(* Logix 5000 project; controller Ceca_1650T_Press 5069-L306ERM rev 32.11; software revision 32.02; part 2 of 3 *)
(* tags used below, declared in another part *)
   STATUS_MESSAGE : STRING;
   AUTO_CYCLE_ENABLED : BOOL;   // M0014 HMI SELECTION
   AUTO_LOWER_LIMIT : BOOL;   // ENCODER SIGNAL B0155
   AUTO_ONE_CYCLE_ENABLED : BOOL;   // M0013 HMI SELECTION
   AUTO_RESET_ALLOWED : BOOL;   // M003E
   AUTO_UPPER_LIMIT : BOOL;   // ENCODER SIGNAL B0151
   BLANKING_OFF_SIGNAL : TIMER;   // T0018
   BLANKING_PS_ENABLED : BOOL;   // M0018
   BOLSTER_CLAMP_ON : BOOL;   // M0006
   BOLSTER_IN_LIMIT : BOOL;   // B000E
   BOLSTER_TOUCH_LIMIT_1 : BOOL;   // B0014
   BOLSTER_TOUCH_LIMIT_2 : BOOL;   // B0015
   BOTH_DIE_CUSHIONS_DOWN : BOOL;   // M0036
   CANCEL_CYLINDER_LOWER_LIMIT : BOOL;   // B000A
   DEBOUNCE_TIMER_LOCKING_OFF : TIMER;   // T0005
   DEBOUNCE_TIMER_LOCKING_OFF_COMPLETE : TIMER;   // T0006
   DECOMPRESSION : BOOL;   // M006D
   DIE_CUSHION_2_PAD_SELECT_RL : BOOL;   // M001D
   DIE_CUSHION_PB_OFF_STATE : BOOL;   // M003F
   DIE_DRAWRIC_CYLINDER_UPPER_PS : BOOL;   // B0018
   DIE_DRAWRIC_DECOMPRESSION_VALVE : BOOL;   // B0056
   DIE_DRAWRIC_DOWN : BOOL;   // M004F
   DIE_DRAWRIC_ON_SELECT : BOOL;   // B0145 HMI BUTTON
   DIE_DRAWRIC_POWER_ASSIST_VALVE : BOOL;   // B0057
   DIE_DRAWRIC_UP : BOOL;   // M004E
   DIE_DRAWRIC_UP_1 : BOOL;   // M007E
   DIE_DRAWRIC_UP_COMPLETE : BOOL;   // M007F
   DIE_DRAWRIC_UP_MEM : TIMER;   // T0019
   DRAW_BLANKING_NOT_SELECT : BOOL;   // M0017
   DRAW_UP_ASSIST : BOOL;   // M007C
   DRAW_UP_ASSIST_COMPLETE : BOOL;   // M007D
   DRAWING_LS_ENABLED : BOOL;   // M0016
   ENABLE_1000T : BOOL;   // HMI BUTTON/RECIPE
   ENABLE_1500T : BOOL;   // HMI BUTTON/RECIPE
   ENABLE_500T : BOOL;   // HMI BUTTON/RECIPE
   FILTER_CHOKER : BOOL;   // B001A
   FILTER_CLOGGED_DELAY : TIMER;   // T0003
   FILTER_CLOGGED_FAULT : BOOL;   // M0023
   FRONT_SHUTTER_SAFETY : BOOL;   // M002A
   INCH_ENABLED : BOOL;   // M0012 HMI SELECTION
   INCHING_SELECTED : BOOL;   // HMI BUTTON/SELECTION B0100
   LOCKING_OFF : BOOL;   // M0004
   LOCKING_OFF_ASSIST : BOOL;   // M0032
   LOCKING_OFF_COMPLETE : BOOL;   // M0033
   LOCKING_OFF_LIMIT : BOOL;   // B0007
   LOCKING_OFF_MEMORY : BOOL;   // M0031
   LOCKING_OFF_VALVE : BOOL;   // B0058
   LOCKING_ON : BOOL;   // M0005
   LOCKING_ON_LIMIT : BOOL;   // B0008
   LUBE_LEVEL_DELAY : TIMER;   // T0002
   LUBE_LEVEL_FAULT : BOOL;   // M0022
   LUBRICATION_FAULT : BOOL;   // M0020
   LUBRICATION_OIL_LEVEL_DETECT : BOOL;   // B001F
   LUBRICATION_PRESSURE_DETECT : BOOL;   // B0017
   M_PRESS_DOWN : BOOL;   // M006A
   M_PRESS_DOWN_COMPLETE : BOOL;   // M006C
   M_PRESS_DOWN_COMPLETE_TIMER : TIMER;   // T0012
   M_PRESS_UP : BOOL;   // M006E
   M_PRESS_UP_COMPLETE : BOOL;   // M006F
   MAIN_DOWN_VALVE : BOOL;   // B0041
   MAIN_DOWN_VALVE_1000_TON : BOOL;   // B0043
   MAIN_DOWN_VALVE_500_TON : BOOL;   // B0042
   MAIN_LOWER_ASSIST_LIMIT : BOOL;   // B0026
   MAIN_LOWER_LIMIT : BOOL;   // B0002
   MAIN_NO_LOAD_VALVE : BOOL;   // B0046
   MAIN_POWER_HOLDING_VALVE : BOOL;   // B0045
   MAIN_PRESS_CONDITION_DOWN : BOOL;   // M0039
   MAIN_PRESS_CONDITION_UP : BOOL;   // M0038
   MAIN_PRESS_DOWN : BOOL;   // M0045
   MAIN_PRESS_DOWN_ASSIST : BOOL;   // M0044
   MAIN_PRESS_NO_PRESSURE_DOWN : BOOL;   // M0047
   MAIN_PRESS_PRESSURE_DETECT : BOOL;   // B0016
   MAIN_PRESS_SLOW_DOWN : BOOL;   // M0046
   MAIN_PRESS_SLOW_DOWN_SIGNAL : BOOL;   // M0030
   MAIN_PRESS_SLOW_UP : BOOL;   // M0042
   MAIN_PRESS_UP : BOOL;   // M0041
   MAIN_PRESS_UP_ASSIST : BOOL;   // M0040
   MAIN_SLOW_DOWN_VALVE : BOOL;   // B0044
   MAIN_UP_VALVE : BOOL;   // B0040
   MAIN_UPPER_LIMIT : BOOL;   // B0000
   MOVEMENT_CONFIRMED : BOOL;   // M0064 M0065 M0066
   NO_PRESSUE_DOWN_PB : BOOL;   // B010D HMI BUTTON
   OIL_TEMP_TOO_HIGH : BOOL;   // B0143
   OIL_TEMPERATURE_FAULT : BOOL;   // M0025
   OIL_WORKING_LEVEL_FAULT : BOOL;   // M0021
   OPERATION_ON : BOOL;   // B0020
   PREFILL_VALVE_OPEN_VALVE : BOOL;   // B0047
   PREFILL_VALVE_OPEN_VALVE_2 : BOOL;   // B0066
   PRESS_AUTO_CYCLE_SELECT_CONDITION : BOOL;   // M0060
   PRESS_AUTO_RUN : BOOL;   // M0069
   PRESS_AUTO_START_POSITION : BOOL;   // M0063
   PRESS_AUTO_START_POSITION_ASSIST : BOOL;   // M0062
   PRESS_HAS_A_FAULT : BOOL;   // M0027
   PRESS_HAS_A_FAULT_2 : BOOL;   // M0028
   PRESS_HOLDING_TIME : BOOL;   // M006B
   PRESS_HOLDING_TIMER : TIMER;   // PRESS HOLDING TIMER
   PRESS_READY_CONFIRM : BOOL;   // M0043
   PUMP_ON_DELAY_CHECK : TIMER;   // T0000
   PUMP_RUN : BOOL;   // B0021
   RESET_PB : BOOL;   // HMI RESET PB
   RESETTING_CONFIRMATION : BOOL;   // M0061
   SAFETY_BAR_OPENED : BOOL;   // B000B
   SLIDE_DOWN_PB : BOOL;   // B010B HMI BUTTON
   SLIDE_SLOW_DOWN_PB : BOOL;   // B010C HMI BUTTON
   SLIDE_SLOW_DOWN_SIGNAL : BOOL;   // B0154 ENCODER SIGNAL
   SLIDE_SLOW_UP_PB : BOOL;   // B010A HMI BUTTON
   SLIDE_UP_PB : BOOL;   // HMI BUTTON B0109
   TIMER_OFF_DELAY_1500T : TIMER;   // T0017
   TIMER_OFF_DELAY_500T : TIMER;   // T0016
   WORKING_LEVEL_DELAY_CHECK : TIMER;   // T0001
   WORKING_OIL_LEVEL_DETECT : BOOL;   // B0025
(* MainProgram, continued *)

ROUTINE Draw   (* ladder *)
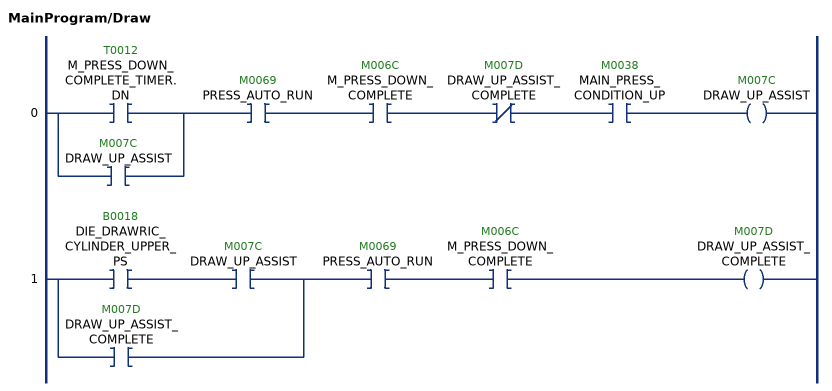
   0: [XIC(M_PRESS_DOWN_COMPLETE_TIMER.DN) ,XIC(DRAW_UP_ASSIST) ]XIC(PRESS_AUTO_RUN)XIC(M_PRESS_DOWN_COMPLETE)XIO(DRAW_UP_ASSIST_COMPLETE)XIC(MAIN_PRESS_CONDITION_UP)OTE(DRAW_UP_ASSIST);
   1: [XIC(DIE_DRAWRIC_CYLINDER_UPPER_PS) XIC(DRAW_UP_ASSIST) ,XIC(DRAW_UP_ASSIST_COMPLETE) ]XIC(PRESS_AUTO_RUN)XIC(M_PRESS_DOWN_COMPLETE)OTE(DRAW_UP_ASSIST_COMPLETE);
END_ROUTINE

ROUTINE Drawric   (* ladder *)
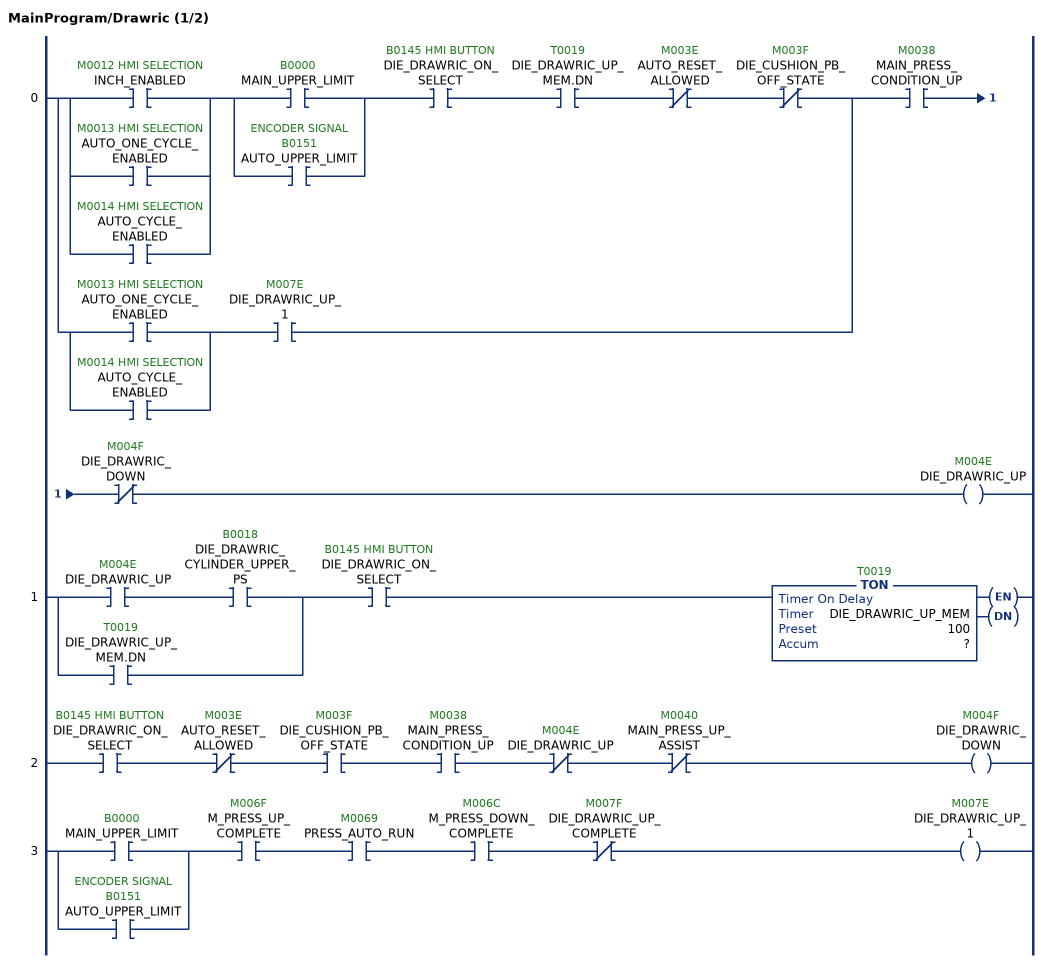
   0: [[XIC(INCH_ENABLED) ,XIC(AUTO_ONE_CYCLE_ENABLED) ,XIC(AUTO_CYCLE_ENABLED) ] [XIC(MAIN_UPPER_LIMIT) ,XIC(AUTO_UPPER_LIMIT) ] XIC(DIE_DRAWRIC_ON_SELECT) XIC(DIE_DRAWRIC_UP_MEM.DN) XIO(AUTO_RESET_ALLOWED) XIO(DIE_CUSHION_PB_OFF_STATE) ,[XIC(AUTO_ONE_CYCLE_ENABLED) ,XIC(AUTO_CYCLE_ENABLED) ] XIC(DIE_DRAWRIC_UP_1) ]XIC(MAIN_PRESS_CONDITION_UP)XIO(DIE_DRAWRIC_DOWN)OTE(DIE_DRAWRIC_UP);
   1: [XIC(DIE_DRAWRIC_UP) XIC(DIE_DRAWRIC_CYLINDER_UPPER_PS) ,XIC(DIE_DRAWRIC_UP_MEM.DN) ]XIC(DIE_DRAWRIC_ON_SELECT)TON(DIE_DRAWRIC_UP_MEM,?,?);
   2: XIC(DIE_DRAWRIC_ON_SELECT)XIO(AUTO_RESET_ALLOWED)XIC(DIE_CUSHION_PB_OFF_STATE)XIC(MAIN_PRESS_CONDITION_UP)XIO(DIE_DRAWRIC_UP)XIO(MAIN_PRESS_UP_ASSIST)OTE(DIE_DRAWRIC_DOWN);
   3: [XIC(MAIN_UPPER_LIMIT) ,XIC(AUTO_UPPER_LIMIT) ]XIC(M_PRESS_UP_COMPLETE)XIC(PRESS_AUTO_RUN)XIC(M_PRESS_DOWN_COMPLETE)XIO(DIE_DRAWRIC_UP_COMPLETE)OTE(DIE_DRAWRIC_UP_1);
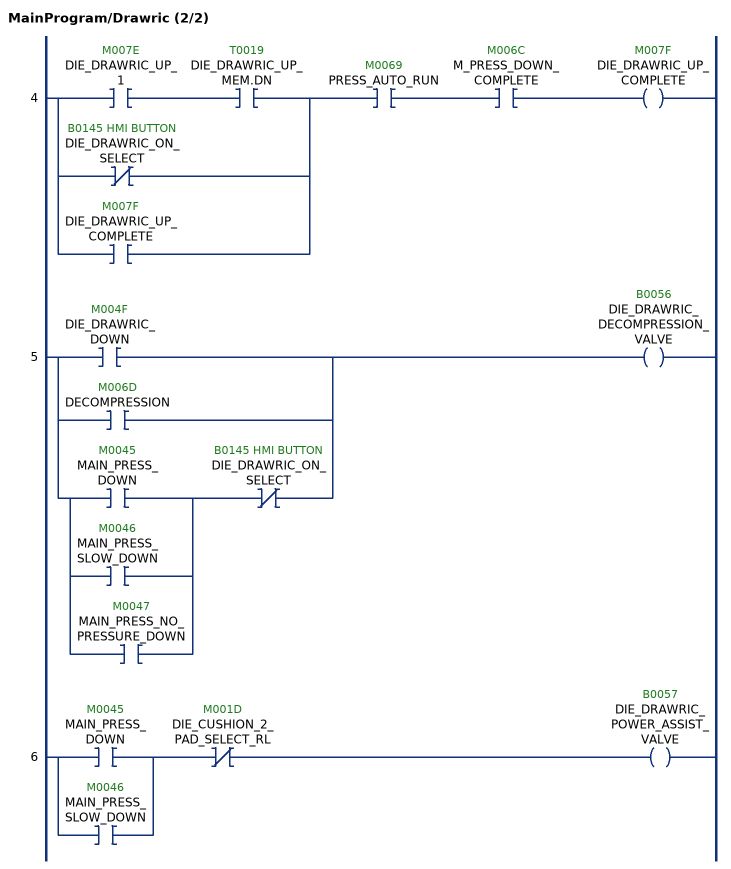
   4: [XIC(DIE_DRAWRIC_UP_1) XIC(DIE_DRAWRIC_UP_MEM.DN) ,XIO(DIE_DRAWRIC_ON_SELECT) ,XIC(DIE_DRAWRIC_UP_COMPLETE) ]XIC(PRESS_AUTO_RUN)XIC(M_PRESS_DOWN_COMPLETE)OTE(DIE_DRAWRIC_UP_COMPLETE);
   5: [XIC(DIE_DRAWRIC_DOWN) ,XIC(DECOMPRESSION) ,[XIC(MAIN_PRESS_DOWN) ,XIC(MAIN_PRESS_SLOW_DOWN) ,XIC(MAIN_PRESS_NO_PRESSURE_DOWN) ] XIO(DIE_DRAWRIC_ON_SELECT) ]OTE(DIE_DRAWRIC_DECOMPRESSION_VALVE);
   6: [XIC(MAIN_PRESS_DOWN) ,XIC(MAIN_PRESS_SLOW_DOWN) ]XIO(DIE_CUSHION_2_PAD_SELECT_RL)OTE(DIE_DRAWRIC_POWER_ASSIST_VALVE);
END_ROUTINE

ROUTINE Faults   (* ladder *)
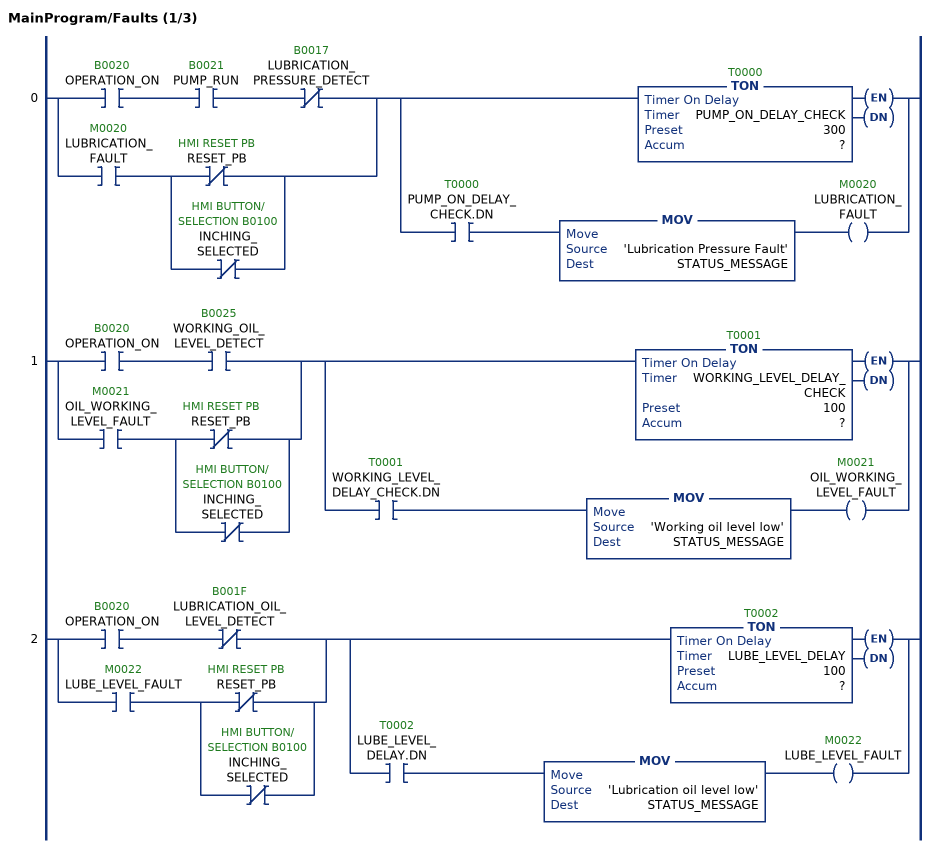
   0: [XIC(OPERATION_ON) XIC(PUMP_RUN) XIO(LUBRICATION_PRESSURE_DETECT) ,XIC(LUBRICATION_FAULT) [XIO(RESET_PB) ,XIO(INCHING_SELECTED) ] ][TON(PUMP_ON_DELAY_CHECK,?,?) ,XIC(PUMP_ON_DELAY_CHECK.DN) MOV('Lubrication Pressure Fault',STATUS_MESSAGE) OTE(LUBRICATION_FAULT) ];
   1: [XIC(OPERATION_ON) XIC(WORKING_OIL_LEVEL_DETECT) ,XIC(OIL_WORKING_LEVEL_FAULT) [XIO(RESET_PB) ,XIO(INCHING_SELECTED) ] ][TON(WORKING_LEVEL_DELAY_CHECK,?,?) ,XIC(WORKING_LEVEL_DELAY_CHECK.DN) MOV('Working oil level low',STATUS_MESSAGE) OTE(OIL_WORKING_LEVEL_FAULT) ];
   2: [XIC(OPERATION_ON) XIO(LUBRICATION_OIL_LEVEL_DETECT) ,XIC(LUBE_LEVEL_FAULT) [XIO(RESET_PB) ,XIO(INCHING_SELECTED) ] ][TON(LUBE_LEVEL_DELAY,?,?) ,XIC(LUBE_LEVEL_DELAY.DN) MOV('Lubrication oil level low',STATUS_MESSAGE) OTE(LUBE_LEVEL_FAULT) ];
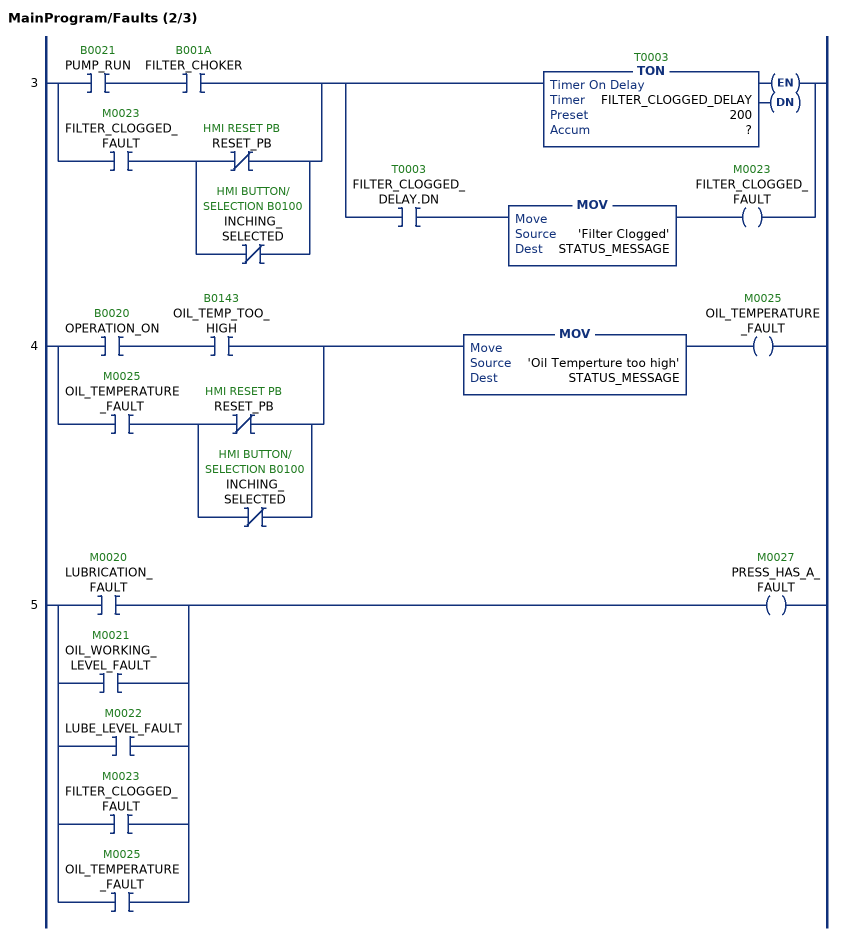
   3: [XIC(PUMP_RUN) XIC(FILTER_CHOKER) ,XIC(FILTER_CLOGGED_FAULT) [XIO(RESET_PB) ,XIO(INCHING_SELECTED) ] ][TON(FILTER_CLOGGED_DELAY,?,?) ,XIC(FILTER_CLOGGED_DELAY.DN) MOV('Filter Clogged',STATUS_MESSAGE) OTE(FILTER_CLOGGED_FAULT) ];
   4: [XIC(OPERATION_ON) XIC(OIL_TEMP_TOO_HIGH) ,XIC(OIL_TEMPERATURE_FAULT) [XIO(RESET_PB) ,XIO(INCHING_SELECTED) ] ]MOV('Oil Temperture too high',STATUS_MESSAGE)OTE(OIL_TEMPERATURE_FAULT);
   5: [XIC(LUBRICATION_FAULT) ,XIC(OIL_WORKING_LEVEL_FAULT) ,XIC(LUBE_LEVEL_FAULT) ,XIC(FILTER_CLOGGED_FAULT) ,XIC(OIL_TEMPERATURE_FAULT) ]OTE(PRESS_HAS_A_FAULT);
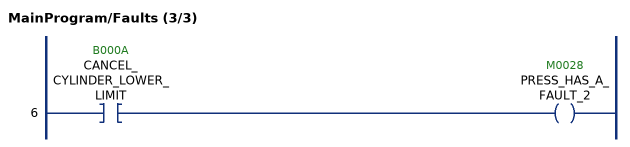
   6: XIC(CANCEL_CYLINDER_LOWER_LIMIT)OTE(PRESS_HAS_A_FAULT_2);
END_ROUTINE

ROUTINE Inputs   (* ladder *)
   0: ;
END_ROUTINE

ROUTINE Locking   (* ladder *)
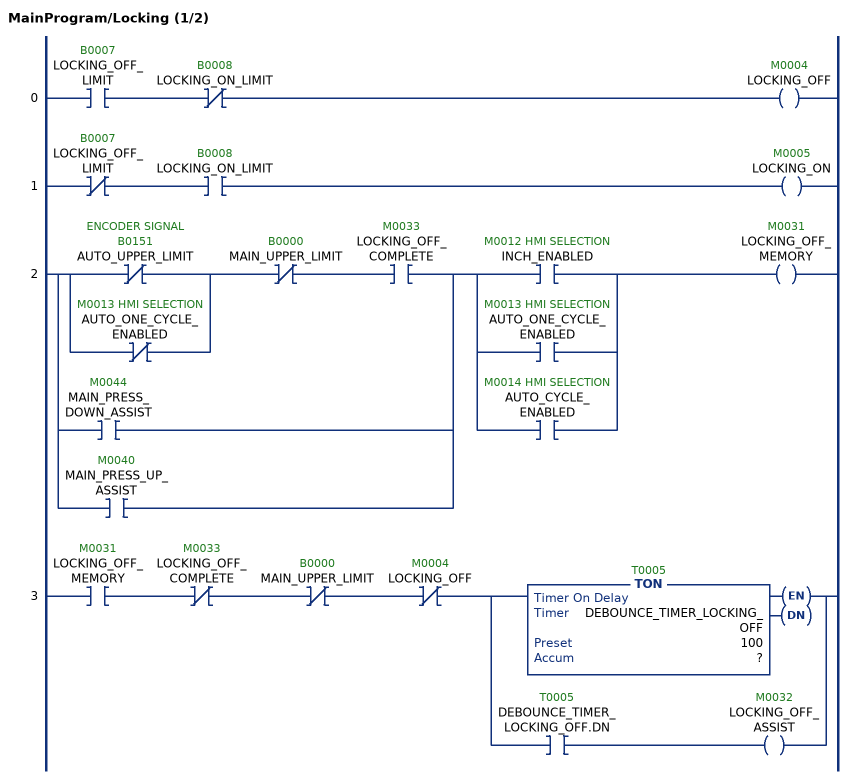
   0: XIC(LOCKING_OFF_LIMIT)XIO(LOCKING_ON_LIMIT)OTE(LOCKING_OFF);
   1: XIO(LOCKING_OFF_LIMIT)XIC(LOCKING_ON_LIMIT)OTE(LOCKING_ON);
   2: [[XIO(AUTO_UPPER_LIMIT) ,XIO(AUTO_ONE_CYCLE_ENABLED) ] XIO(MAIN_UPPER_LIMIT) XIC(LOCKING_OFF_COMPLETE) ,XIC(MAIN_PRESS_DOWN_ASSIST) ,XIC(MAIN_PRESS_UP_ASSIST) ][XIC(INCH_ENABLED) ,XIC(AUTO_ONE_CYCLE_ENABLED) ,XIC(AUTO_CYCLE_ENABLED) ]OTE(LOCKING_OFF_MEMORY);
   3: XIC(LOCKING_OFF_MEMORY)XIO(LOCKING_OFF_COMPLETE)XIO(MAIN_UPPER_LIMIT)XIO(LOCKING_OFF)[TON(DEBOUNCE_TIMER_LOCKING_OFF,?,?) ,XIC(DEBOUNCE_TIMER_LOCKING_OFF.DN) OTE(LOCKING_OFF_ASSIST) ];
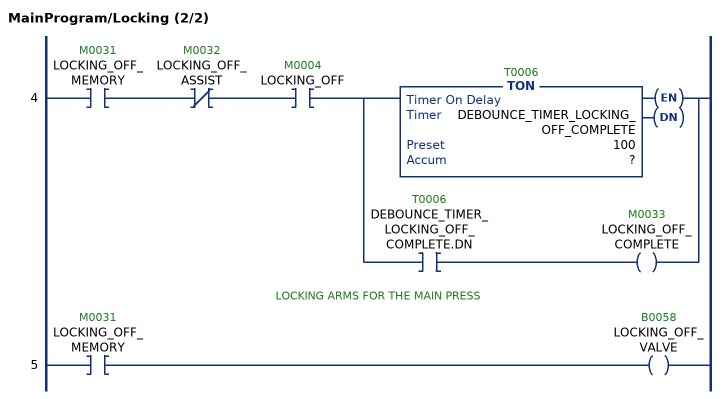
   4: XIC(LOCKING_OFF_MEMORY)XIO(LOCKING_OFF_ASSIST)XIC(LOCKING_OFF)[TON(DEBOUNCE_TIMER_LOCKING_OFF_COMPLETE,?,?) ,XIC(DEBOUNCE_TIMER_LOCKING_OFF_COMPLETE.DN) OTE(LOCKING_OFF_COMPLETE) ];
   // LOCKING ARMS FOR THE MAIN PRESS
   5: XIC(LOCKING_OFF_MEMORY)OTE(LOCKING_OFF_VALVE);
END_ROUTINE

ROUTINE Main_Down   (* ladder *)
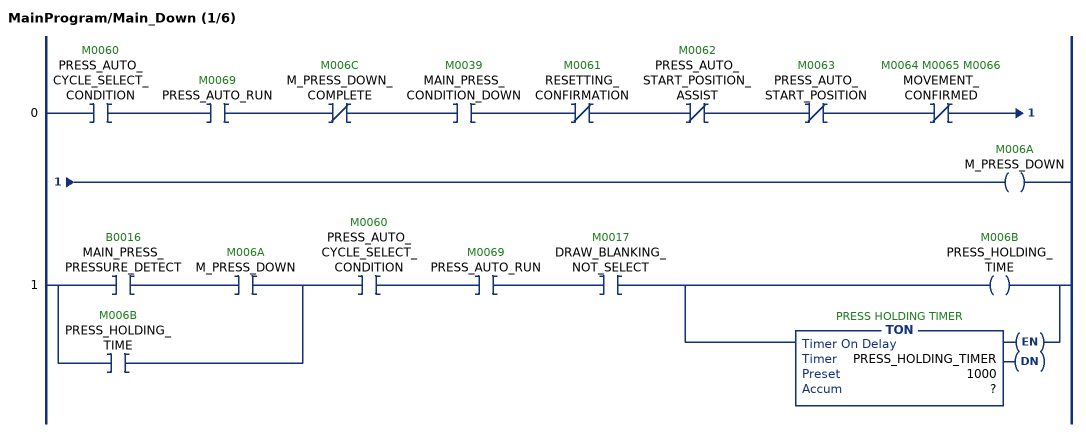
   0: XIC(PRESS_AUTO_CYCLE_SELECT_CONDITION)XIC(PRESS_AUTO_RUN)XIO(M_PRESS_DOWN_COMPLETE)XIC(MAIN_PRESS_CONDITION_DOWN)XIO(RESETTING_CONFIRMATION)XIO(PRESS_AUTO_START_POSITION_ASSIST)XIO(PRESS_AUTO_START_POSITION)XIO(MOVEMENT_CONFIRMED)OTE(M_PRESS_DOWN);
   1: [XIC(MAIN_PRESS_PRESSURE_DETECT) XIC(M_PRESS_DOWN) ,XIC(PRESS_HOLDING_TIME) ]XIC(PRESS_AUTO_CYCLE_SELECT_CONDITION)XIC(PRESS_AUTO_RUN)XIC(DRAW_BLANKING_NOT_SELECT)[OTE(PRESS_HOLDING_TIME) ,TON(PRESS_HOLDING_TIMER,?,?) ];
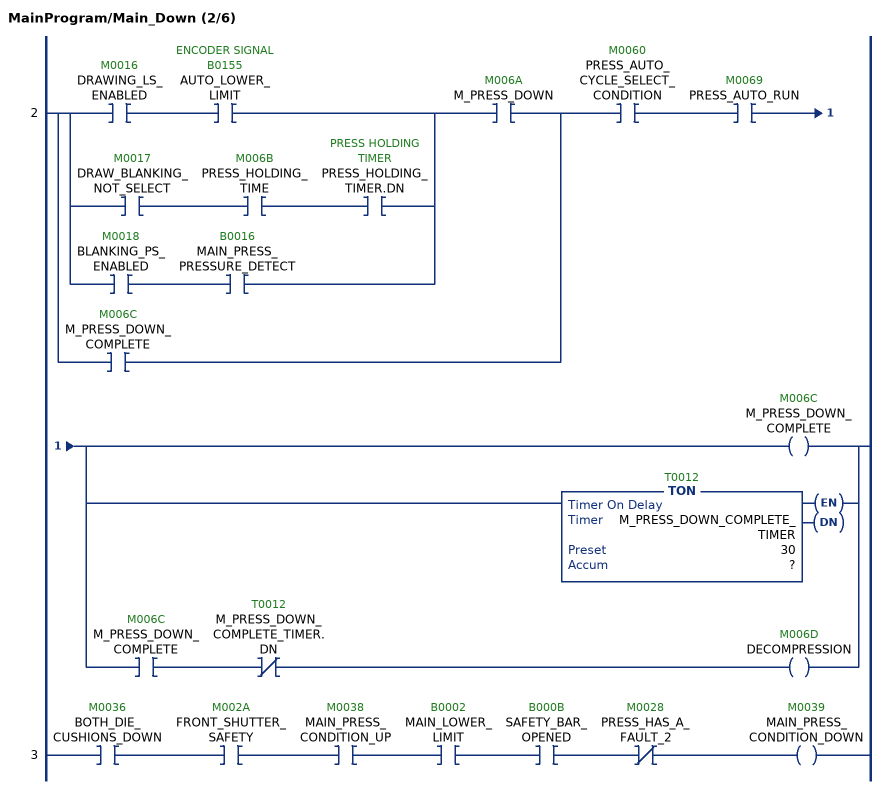
   2: [[XIC(DRAWING_LS_ENABLED) XIC(AUTO_LOWER_LIMIT) ,XIC(DRAW_BLANKING_NOT_SELECT) XIC(PRESS_HOLDING_TIME) XIC(PRESS_HOLDING_TIMER.DN) ,XIC(BLANKING_PS_ENABLED) XIC(MAIN_PRESS_PRESSURE_DETECT) ] XIC(M_PRESS_DOWN) ,XIC(M_PRESS_DOWN_COMPLETE) ]XIC(PRESS_AUTO_CYCLE_SELECT_CONDITION)XIC(PRESS_AUTO_RUN)[OTE(M_PRESS_DOWN_COMPLETE) ,TON(M_PRESS_DOWN_COMPLETE_TIMER,?,?) ,XIC(M_PRESS_DOWN_COMPLETE) XIO(M_PRESS_DOWN_COMPLETE_TIMER.DN) OTE(DECOMPRESSION) ];
   3: XIC(BOTH_DIE_CUSHIONS_DOWN)XIC(FRONT_SHUTTER_SAFETY)XIC(MAIN_PRESS_CONDITION_UP)XIC(MAIN_LOWER_LIMIT)XIC(SAFETY_BAR_OPENED)XIO(PRESS_HAS_A_FAULT_2)OTE(MAIN_PRESS_CONDITION_DOWN);
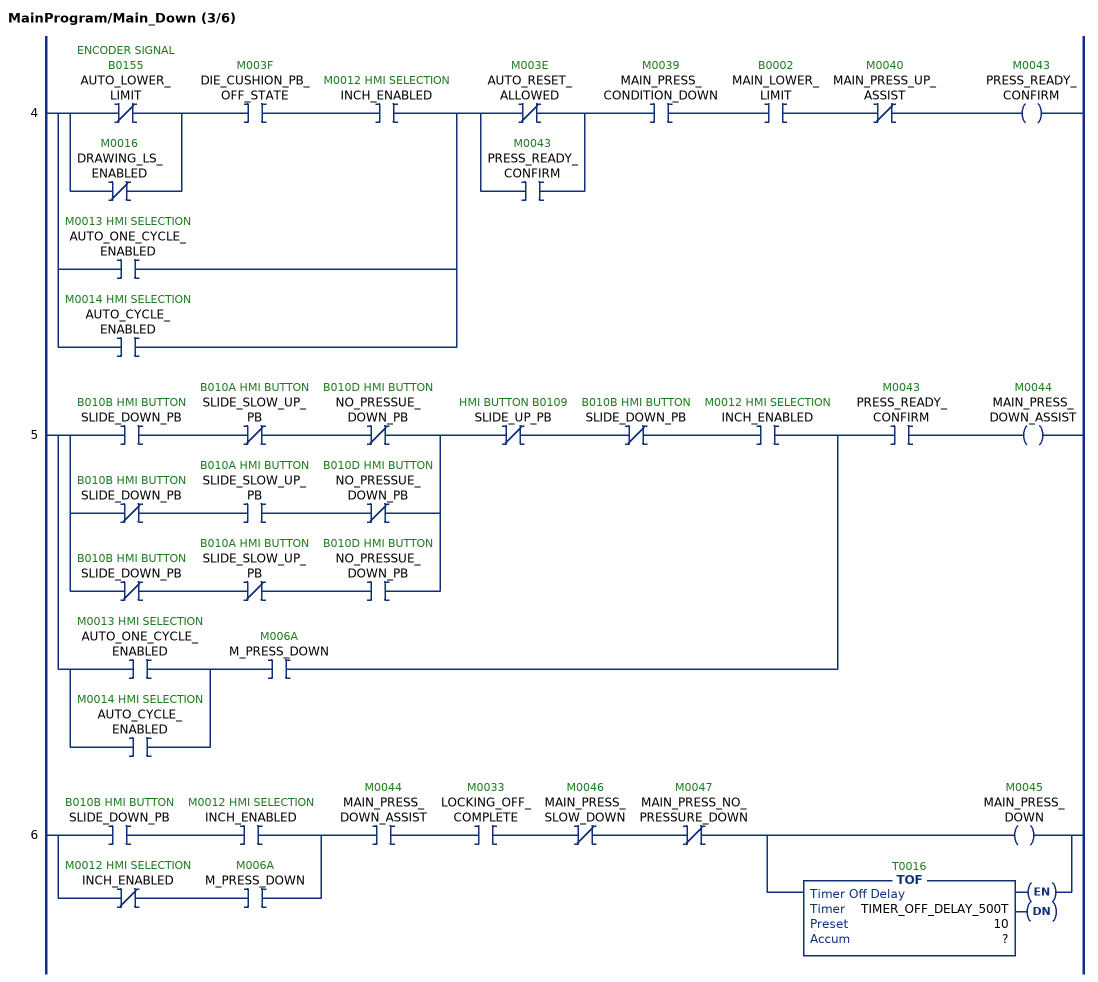
   4: [[XIO(AUTO_LOWER_LIMIT) ,XIO(DRAWING_LS_ENABLED) ] XIC(DIE_CUSHION_PB_OFF_STATE) XIC(INCH_ENABLED) ,XIC(AUTO_ONE_CYCLE_ENABLED) ,XIC(AUTO_CYCLE_ENABLED) ][XIO(AUTO_RESET_ALLOWED) ,XIC(PRESS_READY_CONFIRM) ]XIC(MAIN_PRESS_CONDITION_DOWN)XIC(MAIN_LOWER_LIMIT)XIO(MAIN_PRESS_UP_ASSIST)OTE(PRESS_READY_CONFIRM);
   5: [[XIC(SLIDE_DOWN_PB) XIO(SLIDE_SLOW_UP_PB) XIO(NO_PRESSUE_DOWN_PB) ,XIO(SLIDE_DOWN_PB) XIC(SLIDE_SLOW_UP_PB) XIO(NO_PRESSUE_DOWN_PB) ,XIO(SLIDE_DOWN_PB) XIO(SLIDE_SLOW_UP_PB) XIC(NO_PRESSUE_DOWN_PB) ] XIO(SLIDE_UP_PB) XIO(SLIDE_DOWN_PB) XIC(INCH_ENABLED) ,[XIC(AUTO_ONE_CYCLE_ENABLED) ,XIC(AUTO_CYCLE_ENABLED) ] XIC(M_PRESS_DOWN) ]XIC(PRESS_READY_CONFIRM)OTE(MAIN_PRESS_DOWN_ASSIST);
   6: [XIC(SLIDE_DOWN_PB) XIC(INCH_ENABLED) ,XIO(INCH_ENABLED) XIC(M_PRESS_DOWN) ]XIC(MAIN_PRESS_DOWN_ASSIST)XIC(LOCKING_OFF_COMPLETE)XIO(MAIN_PRESS_SLOW_DOWN)XIO(MAIN_PRESS_NO_PRESSURE_DOWN)[OTE(MAIN_PRESS_DOWN) ,TOF(TIMER_OFF_DELAY_500T,?,?) ];
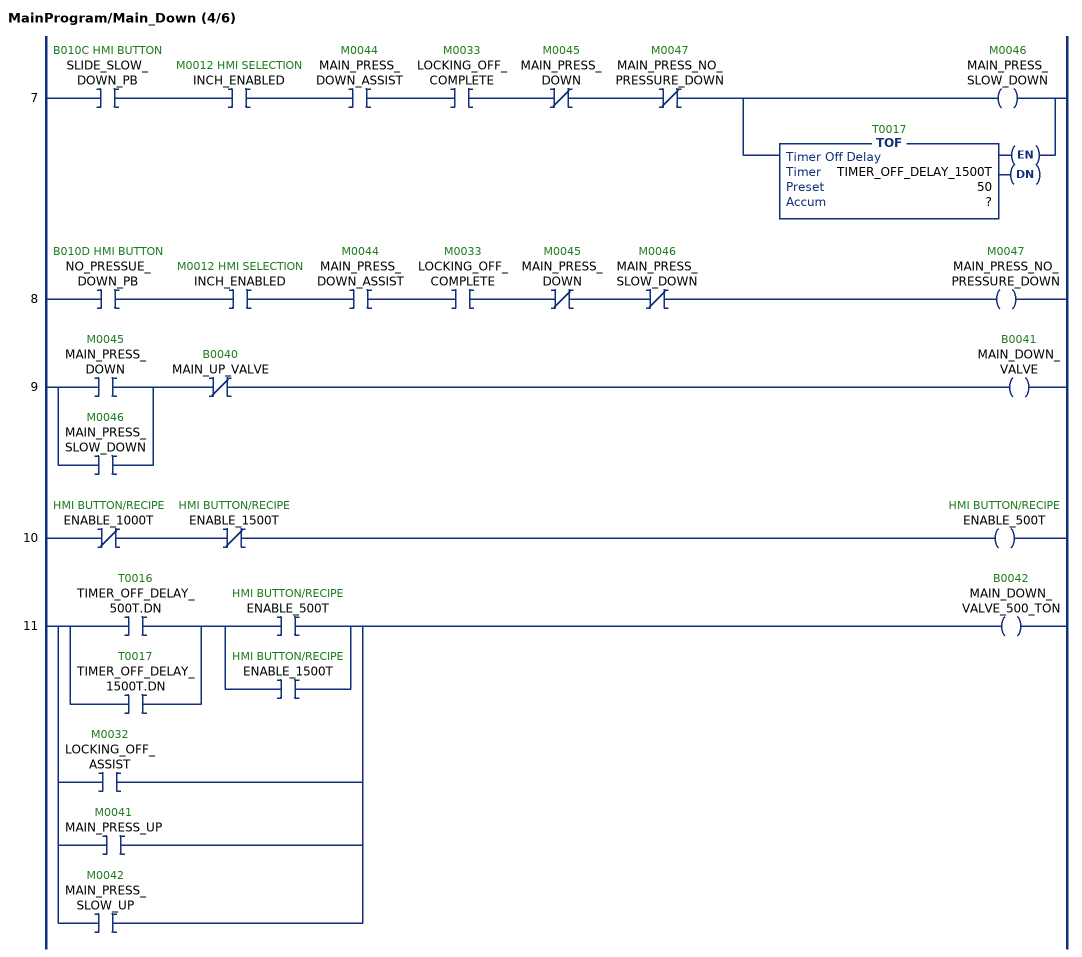
   7: XIC(SLIDE_SLOW_DOWN_PB)XIC(INCH_ENABLED)XIC(MAIN_PRESS_DOWN_ASSIST)XIC(LOCKING_OFF_COMPLETE)XIO(MAIN_PRESS_DOWN)XIO(MAIN_PRESS_NO_PRESSURE_DOWN)[OTE(MAIN_PRESS_SLOW_DOWN) ,TOF(TIMER_OFF_DELAY_1500T,?,?) ];
   8: XIC(NO_PRESSUE_DOWN_PB)XIC(INCH_ENABLED)XIC(MAIN_PRESS_DOWN_ASSIST)XIC(LOCKING_OFF_COMPLETE)XIO(MAIN_PRESS_DOWN)XIO(MAIN_PRESS_SLOW_DOWN)OTE(MAIN_PRESS_NO_PRESSURE_DOWN);
   9: [XIC(MAIN_PRESS_DOWN) ,XIC(MAIN_PRESS_SLOW_DOWN) ]XIO(MAIN_UP_VALVE)OTE(MAIN_DOWN_VALVE);
   10: XIO(ENABLE_1000T)XIO(ENABLE_1500T)OTE(ENABLE_500T);
   11: [[XIC(TIMER_OFF_DELAY_500T.DN) ,XIC(TIMER_OFF_DELAY_1500T.DN) ] [XIC(ENABLE_500T) ,XIC(ENABLE_1500T) ] ,XIC(LOCKING_OFF_ASSIST) ,XIC(MAIN_PRESS_UP) ,XIC(MAIN_PRESS_SLOW_UP) ]OTE(MAIN_DOWN_VALVE_500_TON);
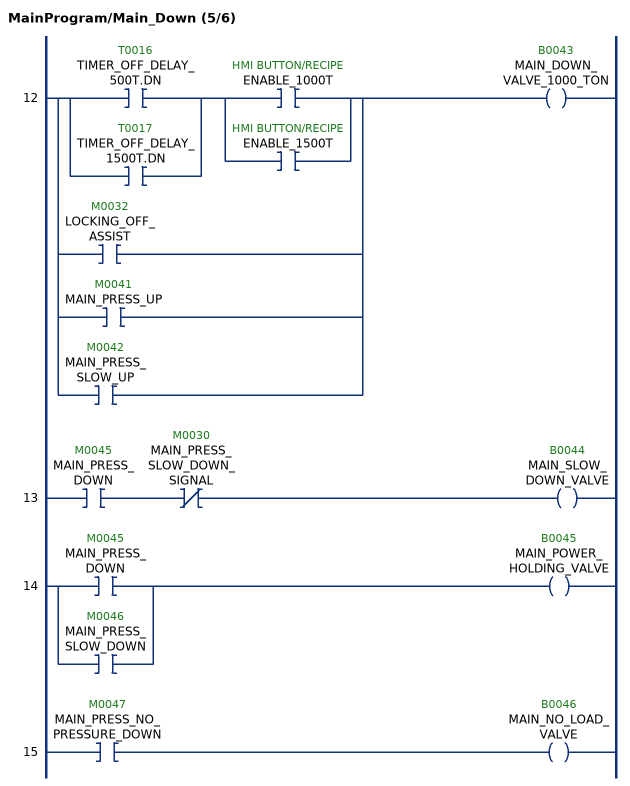
   12: [[XIC(TIMER_OFF_DELAY_500T.DN) ,XIC(TIMER_OFF_DELAY_1500T.DN) ] [XIC(ENABLE_1000T) ,XIC(ENABLE_1500T) ] ,XIC(LOCKING_OFF_ASSIST) ,XIC(MAIN_PRESS_UP) ,XIC(MAIN_PRESS_SLOW_UP) ]OTE(MAIN_DOWN_VALVE_1000_TON);
   13: XIC(MAIN_PRESS_DOWN)XIO(MAIN_PRESS_SLOW_DOWN_SIGNAL)OTE(MAIN_SLOW_DOWN_VALVE);
   14: [XIC(MAIN_PRESS_DOWN) ,XIC(MAIN_PRESS_SLOW_DOWN) ]OTE(MAIN_POWER_HOLDING_VALVE);
   15: XIC(MAIN_PRESS_NO_PRESSURE_DOWN)OTE(MAIN_NO_LOAD_VALVE);
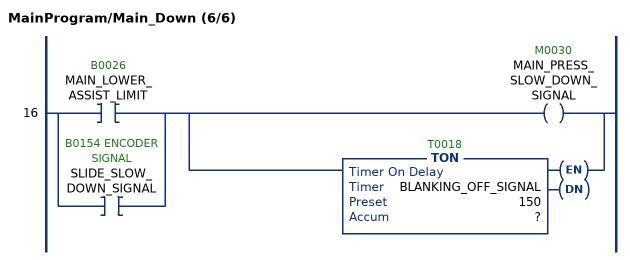
   16: [XIC(MAIN_LOWER_ASSIST_LIMIT) ,XIC(SLIDE_SLOW_DOWN_SIGNAL) ][OTE(MAIN_PRESS_SLOW_DOWN_SIGNAL) ,TON(BLANKING_OFF_SIGNAL,?,?) ];
END_ROUTINE

ROUTINE Main_Up   (* ladder *)
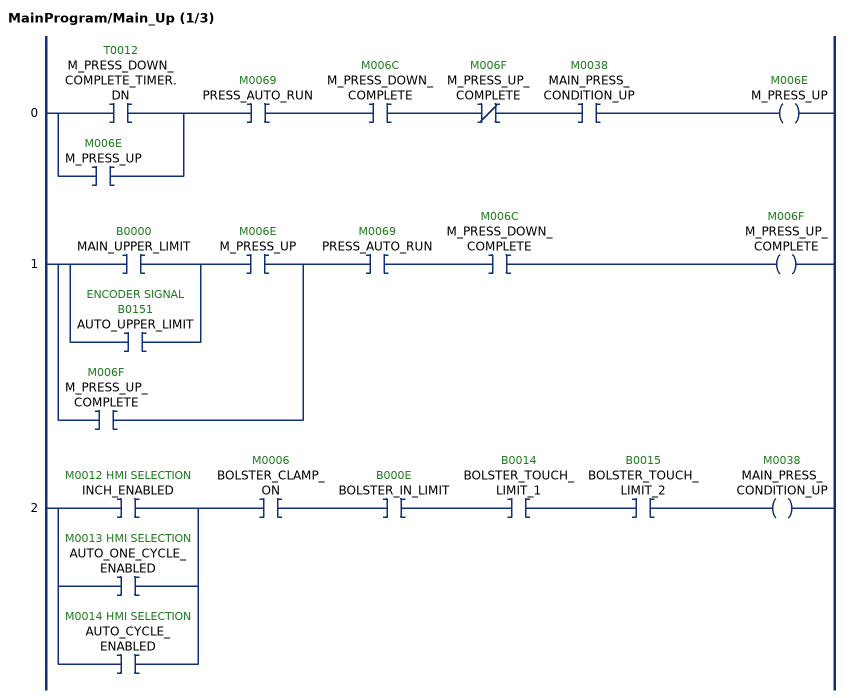
   0: [XIC(M_PRESS_DOWN_COMPLETE_TIMER.DN) ,XIC(M_PRESS_UP) ]XIC(PRESS_AUTO_RUN)XIC(M_PRESS_DOWN_COMPLETE)XIO(M_PRESS_UP_COMPLETE)XIC(MAIN_PRESS_CONDITION_UP)OTE(M_PRESS_UP);
   1: [[XIC(MAIN_UPPER_LIMIT) ,XIC(AUTO_UPPER_LIMIT) ] XIC(M_PRESS_UP) ,XIC(M_PRESS_UP_COMPLETE) ]XIC(PRESS_AUTO_RUN)XIC(M_PRESS_DOWN_COMPLETE)OTE(M_PRESS_UP_COMPLETE);
   2: [XIC(INCH_ENABLED) ,XIC(AUTO_ONE_CYCLE_ENABLED) ,XIC(AUTO_CYCLE_ENABLED) ]XIC(BOLSTER_CLAMP_ON)XIC(BOLSTER_IN_LIMIT)XIC(BOLSTER_TOUCH_LIMIT_1)XIC(BOLSTER_TOUCH_LIMIT_2)OTE(MAIN_PRESS_CONDITION_UP);
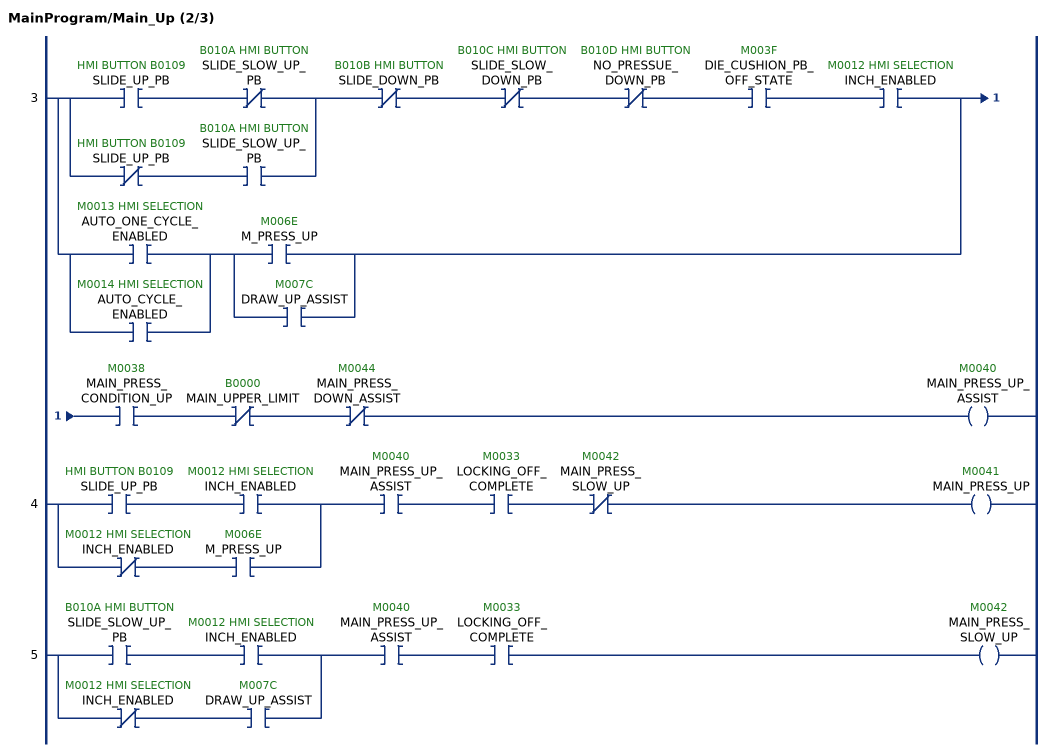
   3: [[XIC(SLIDE_UP_PB) XIO(SLIDE_SLOW_UP_PB) ,XIO(SLIDE_UP_PB) XIC(SLIDE_SLOW_UP_PB) ] XIO(SLIDE_DOWN_PB) XIO(SLIDE_SLOW_DOWN_PB) XIO(NO_PRESSUE_DOWN_PB) XIC(DIE_CUSHION_PB_OFF_STATE) XIC(INCH_ENABLED) ,[XIC(AUTO_ONE_CYCLE_ENABLED) ,XIC(AUTO_CYCLE_ENABLED) ] [XIC(M_PRESS_UP) ,XIC(DRAW_UP_ASSIST) ] ]XIC(MAIN_PRESS_CONDITION_UP)XIO(MAIN_UPPER_LIMIT)XIO(MAIN_PRESS_DOWN_ASSIST)OTE(MAIN_PRESS_UP_ASSIST);
   4: [XIC(SLIDE_UP_PB) XIC(INCH_ENABLED) ,XIO(INCH_ENABLED) XIC(M_PRESS_UP) ]XIC(MAIN_PRESS_UP_ASSIST)XIC(LOCKING_OFF_COMPLETE)XIO(MAIN_PRESS_SLOW_UP)OTE(MAIN_PRESS_UP);
   5: [XIC(SLIDE_SLOW_UP_PB) XIC(INCH_ENABLED) ,XIO(INCH_ENABLED) XIC(DRAW_UP_ASSIST) ]XIC(MAIN_PRESS_UP_ASSIST)XIC(LOCKING_OFF_COMPLETE)OTE(MAIN_PRESS_SLOW_UP);
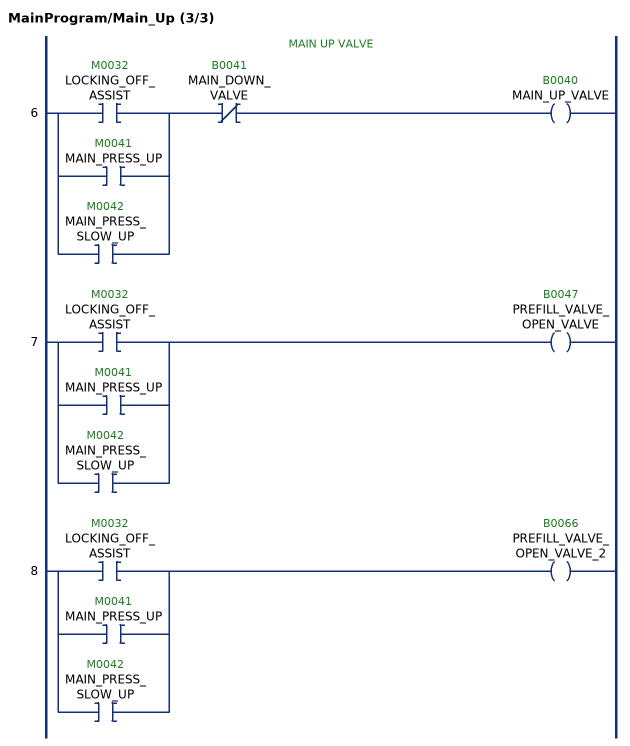
   // MAIN UP VALVE
   6: [XIC(LOCKING_OFF_ASSIST) ,XIC(MAIN_PRESS_UP) ,XIC(MAIN_PRESS_SLOW_UP) ]XIO(MAIN_DOWN_VALVE)OTE(MAIN_UP_VALVE);
   7: [XIC(LOCKING_OFF_ASSIST) ,XIC(MAIN_PRESS_UP) ,XIC(MAIN_PRESS_SLOW_UP) ]OTE(PREFILL_VALVE_OPEN_VALVE);
   8: [XIC(LOCKING_OFF_ASSIST) ,XIC(MAIN_PRESS_UP) ,XIC(MAIN_PRESS_SLOW_UP) ]OTE(PREFILL_VALVE_OPEN_VALVE_2);
END_ROUTINE

ROUTINE MainRoutine   (* ladder *)
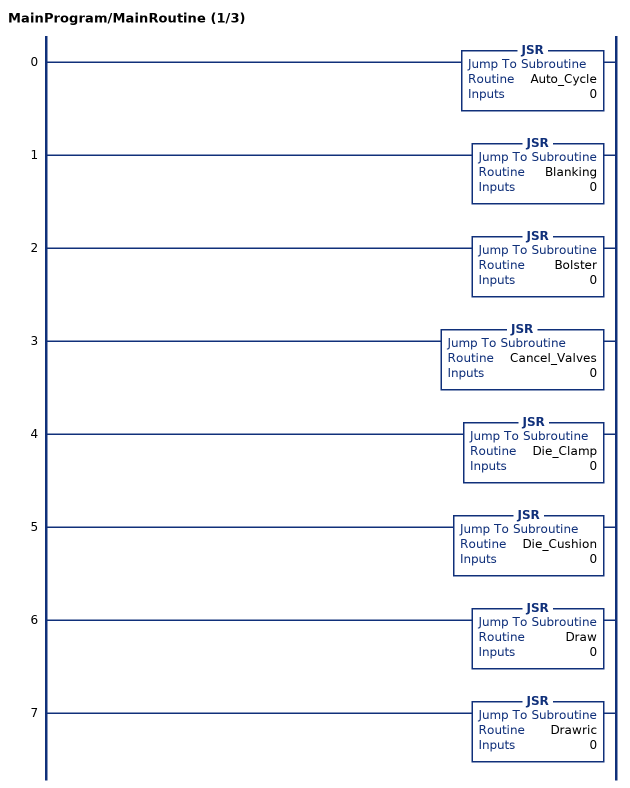
   0: JSR(Auto_Cycle,0);
   1: JSR(Blanking,0);
   2: JSR(Bolster,0);
   3: JSR(Cancel_Valves,0);
   4: JSR(Die_Clamp,0);
   5: JSR(Die_Cushion,0);
   6: JSR(Draw,0);
   7: JSR(Drawric,0);
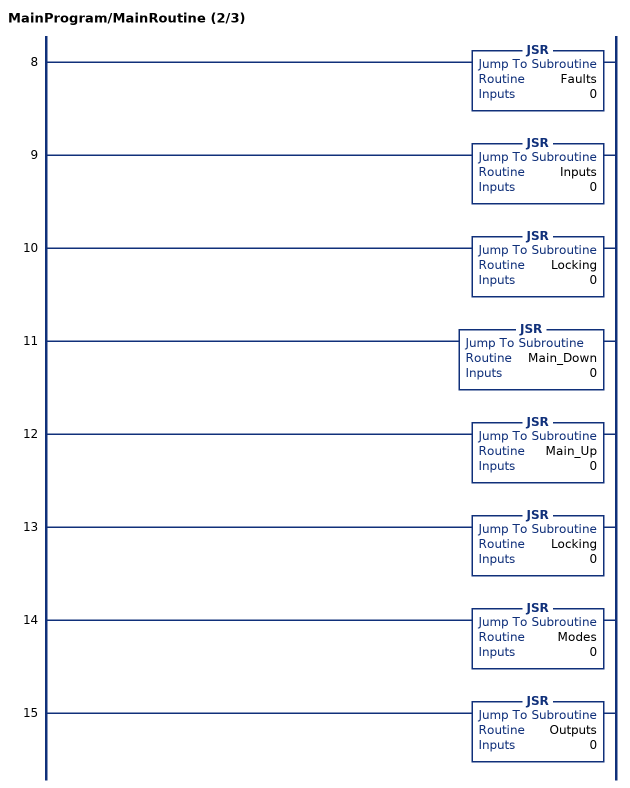
   8: JSR(Faults,0);
   9: JSR(Inputs,0);
   10: JSR(Locking,0);
   11: JSR(Main_Down,0);
   12: JSR(Main_Up,0);
   13: JSR(Locking,0);
   14: JSR(Modes,0);
   15: JSR(Outputs,0);
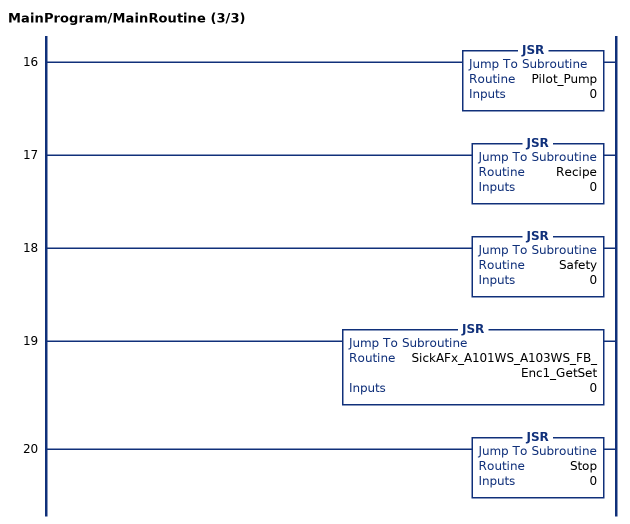
   16: JSR(Pilot_Pump,0);
   17: JSR(Recipe,0);
   18: JSR(Safety,0);
   19: JSR(SickAFx_A101WS_A103WS_FB_Enc1_GetSet,0);
   20: JSR(Stop,0);
END_ROUTINE
